{attribute 'GeneratedUsingTerminal: EP9128-0021-0016'}
{attribute addProperty BoxType "EP9128-0021-0016"}
{attribute addProperty Id "A_0007_EP9128_0021_0017A_0007_EP9128_0021_0017_F9495D48587A_0004_EP9128_0021_0016_2_EP9128_1021EP9128_1FC0878B2"}
{attribute addProperty CRC "3958305985"}
{attribute addProperty Size "589"}
TYPE A_0004_EP9128_0021_0016_EBEEF4C1 EXTENDS EP9128_1FC0878B :
STRUCT
	{attribute addProperty Name "A_0007_EP9128_0021_0017"}
	{attribute addProperty PreviousPort "A_0004(EP9128-0021-0016) : D"}
	A_0007_EP9128_0021_0017 : A_0007_EP9128_0021_0017_F9495D48;
	{attribute addProperty Name "A_0004_EP9128_0021_0016_2_EP9128_1021"}
	{attribute addProperty PreviousPort "A_0004(EP9128-0021-0016) : C"}
	A_0004_EP9128_0021_0016_2_EP9128_1021 : EP9128_1FC0878B;
END_STRUCT
END_TYPE

(* stored: Version 1.2.0.0, ProductVersion 3.1.4024.9
   DUT A_0004_EP9128_0021_0016_EBEEF4C1: Id {b416cb9b-348a-44a3-84d4-25b404741c16} *)
